(* PLC project  *)

CONFIGURATION Empty_Module_21
END_CONFIGURATION
